Fanuc KAREL source: kt00272.KL

-- PROVISIONAL review KL for V940-1; original PC SHA256 fa308cfb13aa77d3fd6c80830f09368b4ab1cf6c302c4592c73b9518576e8650
-- Incomplete behavior may be omitted. Consult companion uncertainty JSON. Do not deploy.
PROGRAM KT00272
%NOLOCKGROUP
VAR
  R2 : REAL
  OUT : BOOLEAN
-- UNRESOLVED_DECL H1 type=002017
BEGIN
  -- V9_ZERO_TABLE_METADATA_HINT layout=0001; no indexed target words; source/name/runtime held
  -- UNRESOLVED_PC offsets 5-19; opcodes 2E,22,9D,33,B4
  -- UNRESOLVED_PC offsets 24-35; opcodes 2E,23
  -- UNRESOLVED_PC offsets 40-64; opcodes 22,9D,33,B3,21,29,64,6D,23
  -- UNRESOLVED_PC offsets 69-73; opcodes 7F
END KT00272
